TYPE ST_Extcontroller_params :
STRUCT
	b_BigEndian				: BOOL;
	b_testComm				: BOOL;
	b_MonitoringEnable		: BOOL := TRUE;
	b_ControlEnable			: BOOL := TRUE;
	w_CommTimeOut			: WORD := 10000; // milli seconds
	TestVars				: ST_PNTest;
	Limits					: ST_ExtController_limits;
END_STRUCT
END_TYPE

(* stored: Version 1.1.0.1, ProductVersion 3.1.4026.18
   DUT ST_Extcontroller_params: Id {ee50a3fe-e09f-410e-bd5d-de2da71f3198} *)
